ABB RAPID module: Operations.mod

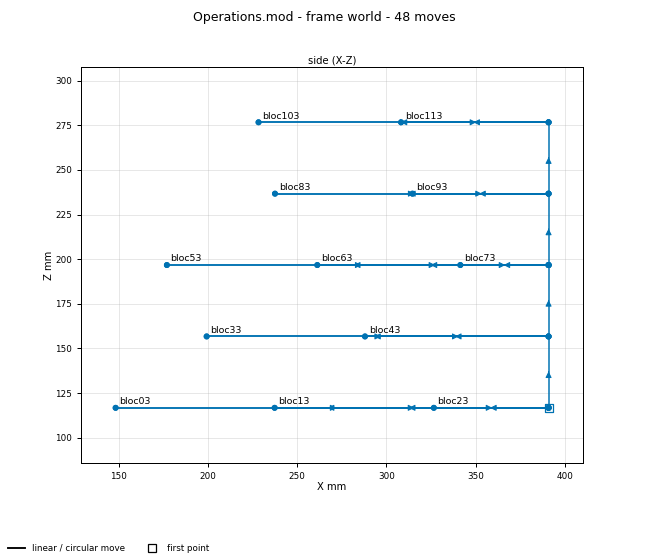
[picture p0: tool path of Operations.mod in frame world, 48 of 49 moves have a stored position in this frame; points joined in program order, loops and branches not executed]
MODULE Operations
 PROC GoHome()
  !
  VAR speeddata HomeSpeed:=[800,100,5000,1000];
  CONST jointtarget HomeTargets0:=[[19.79,37.43,-27.03,0,79.6,44.79],[0,9E9,9E9,9E9,9E9,9E9]];
  MoveAbsJ HomeTargets0,HomeSpeed,z1,EGP_40_N_N_B;
 ENDPROC
 PROC BuildWall()
  !
  VAR zonedata TransportZone:=[FALSE,5,7.5,7.5,0.75,7.5,0.75];
  VAR speeddata PickSpeed:=[60,100,5000,1000];
  CONST robtarget bloc00:=[[16.37,284,122.19],[-0.2706,-0.6533,0.6533,0.2706],[0,0,-1,0],[0,9E9,9E9,9E9,9E9,9E9]];
  CONST robtarget bloc01:=[[-54.35,284,51.47],[-0.2706,-0.6533,0.6533,0.2706],[0,0,-1,0],[0,9E9,9E9,9E9,9E9,9E9]];
  CONST robtarget bloc02:=[[390.93,-147.52,116.72],[0,-0.5676,0.8233,0],[-1,0,-1,0],[0,9E9,9E9,9E9,9E9,9E9]];
  CONST robtarget bloc03:=[[148.33,-147.52,116.72],[0,-0.5676,0.8233,0],[-1,0,-1,0],[0,9E9,9E9,9E9,9E9,9E9]];
  CONST robtarget bloc04:=[[148.33,-263.37,116.72],[0,-0.5676,0.8233,0],[-1,0,-2,0],[0,9E9,9E9,9E9,9E9,9E9]];
  CONST robtarget bloc05:=[[148.33,-263.37,16.72],[0,-0.5676,0.8233,0],[-1,0,-2,0],[0,9E9,9E9,9E9,9E9,9E9]];
  CONST robtarget bloc10:=[[16.37,284,122.19],[-0.2706,-0.6533,0.6533,0.2706],[0,0,-1,0],[0,9E9,9E9,9E9,9E9,9E9]];
  CONST robtarget bloc11:=[[-54.35,284,51.47],[-0.2706,-0.6533,0.6533,0.2706],[0,0,-1,0],[0,9E9,9E9,9E9,9E9,9E9]];
  CONST robtarget bloc12:=[[390.93,-147.52,116.72],[0,-0.6609,0.7505,0],[-1,0,-1,0],[0,9E9,9E9,9E9,9E9,9E9]];
  CONST robtarget bloc13:=[[237.43,-147.52,116.72],[0,-0.6609,0.7505,0],[-1,0,-1,0],[0,9E9,9E9,9E9,9E9,9E9]];
  CONST robtarget bloc14:=[[237.43,-286.18,116.72],[0,-0.6609,0.7505,0],[-1,0,-2,0],[0,9E9,9E9,9E9,9E9,9E9]];
  CONST robtarget bloc15:=[[237.43,-286.18,16.72],[0,-0.6609,0.7505,0],[-1,0,-2,0],[0,9E9,9E9,9E9,9E9,9E9]];
  CONST robtarget bloc20:=[[16.37,284,122.19],[-0.2706,-0.6533,0.6533,0.2706],[0,0,-1,0],[0,9E9,9E9,9E9,9E9,9E9]];
  CONST robtarget bloc21:=[[-54.35,284,51.47],[-0.2706,-0.6533,0.6533,0.2706],[0,0,-1,0],[0,9E9,9E9,9E9,9E9,9E9]];
  CONST robtarget bloc22:=[[390.93,-147.52,116.72],[0,0.7222,-0.6917,0],[-1,0,-1,0],[0,9E9,9E9,9E9,9E9,9E9]];
  CONST robtarget bloc23:=[[326.64,-147.52,116.72],[0,0.7222,-0.6917,0],[-1,0,-2,0],[0,9E9,9E9,9E9,9E9,9E9]];
  CONST robtarget bloc24:=[[326.64,-289.82,116.72],[0,0.7222,-0.6917,0],[-1,0,-2,0],[0,9E9,9E9,9E9,9E9,9E9]];
  CONST robtarget bloc25:=[[326.64,-289.82,16.72],[0,0.7222,-0.6917,0],[-1,0,-2,0],[0,9E9,9E9,9E9,9E9,9E9]];
  CONST robtarget bloc30:=[[16.37,284,122.19],[-0.2706,-0.6533,0.6533,0.2706],[0,0,-1,0],[0,9E9,9E9,9E9,9E9,9E9]];
  CONST robtarget bloc31:=[[-54.35,284,51.47],[-0.2706,-0.6533,0.6533,0.2706],[0,0,-1,0],[0,9E9,9E9,9E9,9E9,9E9]];
  CONST robtarget bloc32:=[[390.93,-147.52,156.72],[0,-0.6058,0.7956,0],[-1,0,-1,0],[0,9E9,9E9,9E9,9E9,9E9]];
  CONST robtarget bloc33:=[[199.33,-147.52,156.72],[0,-0.6058,0.7956,0],[-1,0,-1,0],[0,9E9,9E9,9E9,9E9,9E9]];
  CONST robtarget bloc34:=[[199.33,-268.81,156.72],[0,-0.6058,0.7956,0],[-1,0,-2,0],[0,9E9,9E9,9E9,9E9,9E9]];
  CONST robtarget bloc35:=[[199.33,-268.81,56.72],[0,-0.6058,0.7956,0],[-1,0,-2,0],[0,9E9,9E9,9E9,9E9,9E9]];
  CONST robtarget bloc40:=[[16.37,284,122.19],[-0.2706,-0.6533,0.6533,0.2706],[0,0,-1,0],[0,9E9,9E9,9E9,9E9,9E9]];
  CONST robtarget bloc41:=[[-54.35,284,51.47],[-0.2706,-0.6533,0.6533,0.2706],[0,0,-1,0],[0,9E9,9E9,9E9,9E9,9E9]];
  CONST robtarget bloc42:=[[390.93,-147.52,156.72],[0,-0.6793,0.7339,0],[-1,0,-1,0],[0,9E9,9E9,9E9,9E9,9E9]];
  CONST robtarget bloc43:=[[288.06,-147.52,156.72],[0,-0.6793,0.7339,0],[-1,0,-1,0],[0,9E9,9E9,9E9,9E9,9E9]];
  CONST robtarget bloc44:=[[288.06,-284.33,156.72],[0,-0.6793,0.7339,0],[-1,0,-2,0],[0,9E9,9E9,9E9,9E9,9E9]];
  CONST robtarget bloc45:=[[288.06,-284.33,56.72],[0,-0.6793,0.7339,0],[-1,0,-2,0],[0,9E9,9E9,9E9,9E9,9E9]];
  CONST robtarget bloc50:=[[16.37,284,122.19],[-0.2706,-0.6533,0.6533,0.2706],[0,0,-1,0],[0,9E9,9E9,9E9,9E9,9E9]];
  CONST robtarget bloc51:=[[-54.35,284,51.47],[-0.2706,-0.6533,0.6533,0.2706],[0,0,-1,0],[0,9E9,9E9,9E9,9E9,9E9]];
  CONST robtarget bloc52:=[[390.93,-147.52,196.72],[0,-0.5921,0.8058,0],[-1,0,-1,0],[0,9E9,9E9,9E9,9E9,9E9]];
  CONST robtarget bloc53:=[[177.04,-147.52,196.72],[0,-0.5921,0.8058,0],[-1,0,-1,0],[0,9E9,9E9,9E9,9E9,9E9]];
  CONST robtarget bloc54:=[[177.04,-252.96,196.72],[0,-0.5921,0.8058,0],[-1,0,-2,0],[0,9E9,9E9,9E9,9E9,9E9]];
  CONST robtarget bloc55:=[[177.04,-252.96,96.72],[0,-0.5921,0.8058,0],[-1,0,-2,0],[0,9E9,9E9,9E9,9E9,9E9]];
  CONST robtarget bloc60:=[[16.37,284,122.19],[-0.2706,-0.6533,0.6533,0.2706],[0,0,-1,0],[0,9E9,9E9,9E9,9E9,9E9]];
  CONST robtarget bloc61:=[[-54.35,284,51.47],[-0.2706,-0.6533,0.6533,0.2706],[0,0,-1,0],[0,9E9,9E9,9E9,9E9,9E9]];
  CONST robtarget bloc62:=[[390.93,-147.52,196.72],[0,-0.6476,0.762,0],[-1,0,-1,0],[0,9E9,9E9,9E9,9E9,9E9]];
  CONST robtarget bloc63:=[[261.33,-147.52,196.72],[0,-0.6476,0.762,0],[-1,0,-1,0],[0,9E9,9E9,9E9,9E9,9E9]];
  CONST robtarget bloc64:=[[261.33,-272.79,196.72],[0,-0.6476,0.762,0],[-1,0,-2,0],[0,9E9,9E9,9E9,9E9,9E9]];
  CONST robtarget bloc65:=[[261.33,-272.79,96.72],[0,-0.6476,0.762,0],[-1,0,-2,0],[0,9E9,9E9,9E9,9E9,9E9]];
  CONST robtarget bloc70:=[[16.37,284,122.19],[-0.2706,-0.6533,0.6533,0.2706],[0,0,-1,0],[0,9E9,9E9,9E9,9E9,9E9]];
  CONST robtarget bloc71:=[[-54.35,284,51.47],[-0.2706,-0.6533,0.6533,0.2706],[0,0,-1,0],[0,9E9,9E9,9E9,9E9,9E9]];
  CONST robtarget bloc72:=[[390.93,-147.52,196.72],[0,0.7159,-0.6982,0],[-1,0,-1,0],[0,9E9,9E9,9E9,9E9,9E9]];
  CONST robtarget bloc73:=[[341.48,-147.52,196.72],[0,0.7159,-0.6982,0],[-1,0,-1,0],[0,9E9,9E9,9E9,9E9,9E9]];
  CONST robtarget bloc74:=[[341.48,-279.04,196.72],[0,0.7159,-0.6982,0],[-1,0,-2,0],[0,9E9,9E9,9E9,9E9,9E9]];
  CONST robtarget bloc75:=[[341.48,-279.04,96.72],[0,0.7159,-0.6982,0],[-1,0,-2,0],[0,9E9,9E9,9E9,9E9,9E9]];
  CONST robtarget bloc80:=[[16.37,284,122.19],[-0.2706,-0.6533,0.6533,0.2706],[0,0,-1,0],[0,9E9,9E9,9E9,9E9,9E9]];
  CONST robtarget bloc81:=[[-54.35,284,51.47],[-0.2706,-0.6533,0.6533,0.2706],[0,0,-1,0],[0,9E9,9E9,9E9,9E9,9E9]];
  CONST robtarget bloc82:=[[390.93,-147.52,236.72],[0,-0.6442,0.7648,0],[-1,0,-1,0],[0,9E9,9E9,9E9,9E9,9E9]];
  CONST robtarget bloc83:=[[237.62,-147.52,236.72],[0,-0.6442,0.7648,0],[-1,0,-1,0],[0,9E9,9E9,9E9,9E9,9E9]];
  CONST robtarget bloc84:=[[237.62,-258.84,236.72],[0,-0.6442,0.7648,0],[-1,0,-2,0],[0,9E9,9E9,9E9,9E9,9E9]];
  CONST robtarget bloc85:=[[237.62,-258.84,136.72],[0,-0.6442,0.7648,0],[-1,0,-2,0],[0,9E9,9E9,9E9,9E9,9E9]];
  CONST robtarget bloc90:=[[16.37,284,122.19],[-0.2706,-0.6533,0.6533,0.2706],[0,0,-1,0],[0,9E9,9E9,9E9,9E9,9E9]];
  CONST robtarget bloc91:=[[-54.35,284,51.47],[-0.2706,-0.6533,0.6533,0.2706],[0,0,-1,0],[0,9E9,9E9,9E9,9E9,9E9]];
  CONST robtarget bloc92:=[[390.93,-147.52,236.72],[0,-0.6797,0.7335,0],[-1,0,-1,0],[0,9E9,9E9,9E9,9E9,9E9]];
  CONST robtarget bloc93:=[[314.68,-147.52,236.72],[0,-0.6797,0.7335,0],[-1,0,-1,0],[0,9E9,9E9,9E9,9E9,9E9]];
  CONST robtarget bloc94:=[[314.68,-268.74,236.72],[0,-0.6797,0.7335,0],[-1,0,-2,0],[0,9E9,9E9,9E9,9E9,9E9]];
  CONST robtarget bloc95:=[[314.68,-268.74,136.72],[0,-0.6797,0.7335,0],[-1,0,-2,0],[0,9E9,9E9,9E9,9E9,9E9]];
  CONST robtarget bloc100:=[[16.37,284,122.19],[-0.2706,-0.6533,0.6533,0.2706],[0,0,-1,0],[0,9E9,9E9,9E9,9E9,9E9]];
  CONST robtarget bloc101:=[[-54.35,284,51.47],[-0.2706,-0.6533,0.6533,0.2706],[0,0,-1,0],[0,9E9,9E9,9E9,9E9,9E9]];
  CONST robtarget bloc102:=[[390.93,-147.52,276.72],[0,-0.6905,0.7234,0],[-1,0,-1,0],[0,9E9,9E9,9E9,9E9,9E9]];
  CONST robtarget bloc103:=[[228.41,-147.52,276.72],[0,-0.6905,0.7234,0],[-1,0,-2,0],[0,9E9,9E9,9E9,9E9,9E9]];
  CONST robtarget bloc104:=[[228.41,-249.38,276.72],[0,-0.6905,0.7234,0],[-1,0,-2,0],[0,9E9,9E9,9E9,9E9,9E9]];
  CONST robtarget bloc105:=[[228.41,-249.38,176.72],[0,-0.6905,0.7234,0],[-1,0,-2,0],[0,9E9,9E9,9E9,9E9,9E9]];
  CONST robtarget bloc110:=[[16.37,284,122.19],[-0.2706,-0.6533,0.6533,0.2706],[0,0,-1,0],[0,9E9,9E9,9E9,9E9,9E9]];
  CONST robtarget bloc111:=[[-54.35,284,51.47],[-0.2706,-0.6533,0.6533,0.2706],[0,0,-1,0],[0,9E9,9E9,9E9,9E9,9E9]];
  CONST robtarget bloc112:=[[390.93,-147.52,276.72],[0,-0.6849,0.7286,0],[-1,0,-1,0],[0,9E9,9E9,9E9,9E9,9E9]];
  CONST robtarget bloc113:=[[308.27,-147.52,276.72],[0,-0.6849,0.7286,0],[-1,0,-1,0],[0,9E9,9E9,9E9,9E9,9E9]];
  CONST robtarget bloc114:=[[308.27,-253.64,276.72],[0,-0.6849,0.7286,0],[-1,0,-2,0],[0,9E9,9E9,9E9,9E9,9E9]];
  CONST robtarget bloc115:=[[308.27,-253.64,176.72],[0,-0.6849,0.7286,0],[-1,0,-2,0],[0,9E9,9E9,9E9,9E9,9E9]];
  CONST robtarget NNCTarget0:=[[0,0,101],[0,0,1,0],[0,0,1,0],[0,9E9,9E9,9E9,9E9,9E9]];
  CONST robtarget NNCTarget1:=[[0,0,100],[0,0,1,0],[0,0,1,0],[0,9E9,9E9,9E9,9E9,9E9]];
  CONST robtarget NNCTarget2:=[[0,0,15],[0,0,1,0],[0,0,1,0],[0,9E9,9E9,9E9,9E9,9E9]];
  CONST robtarget CalibTarget0:=[[-8.38,284,196.43],[-0.2706,-0.6533,0.6533,0.2706],[0,0,-1,0],[0,9E9,9E9,9E9,9E9,9E9]];
  CONST robtarget CalibTarget1:=[[-100.31,284,104.51],[-0.2706,-0.6533,0.6533,0.2706],[0,0,-1,0],[0,9E9,9E9,9E9,9E9,9E9]];
  VAR speeddata TransportSpeed:=[800,100,5000,1000];
  StartGripper;
  PathAccLim TRUE \AccMax:=0.7, TRUE \DecelMax:=0.7;
  FindBlock EGP_40_N_N_B, NNCTarget0, TransportSpeed;
  TakeBloc NNCTarget1, NNCTarget2, EGP_40_N_N_B, TransportSpeed, PickSpeed, blockWobj;
  GoHome;
  ReleaseBloc CalibTarget0, CalibTarget1, EGP_40_N_N_B, TransportSpeed, PickSpeed, WObj0;
  TakeBloc bloc00, bloc01, EGP_40_N_N_B, TransportSpeed, PickSpeed, WObj0;
  GoHome;
  MoveL bloc02,TransportSpeed,TransportZone,EGP_40_N_N_B\WObj:=WObj0;
  MoveL bloc03,TransportSpeed,TransportZone,EGP_40_N_N_B\WObj:=WObj0;
  ReleaseBloc bloc04, bloc05, EGP_40_N_N_B, TransportSpeed, PickSpeed, WObj0;
  MoveL bloc03,TransportSpeed,TransportZone,EGP_40_N_N_B\WObj:=WObj0;
  MoveL bloc02,TransportSpeed,TransportZone,EGP_40_N_N_B\WObj:=WObj0;
  FindBlock EGP_40_N_N_B, NNCTarget0, TransportSpeed;
  TakeBloc NNCTarget1, NNCTarget2, EGP_40_N_N_B, TransportSpeed, PickSpeed, blockWobj;
  GoHome;
  ReleaseBloc CalibTarget0, CalibTarget1, EGP_40_N_N_B, TransportSpeed, PickSpeed, WObj0;
  TakeBloc bloc10, bloc11, EGP_40_N_N_B, TransportSpeed, PickSpeed, WObj0;
  GoHome;
  MoveL bloc12,TransportSpeed,TransportZone,EGP_40_N_N_B\WObj:=WObj0;
  MoveL bloc13,TransportSpeed,TransportZone,EGP_40_N_N_B\WObj:=WObj0;
  ReleaseBloc bloc14, bloc15, EGP_40_N_N_B, TransportSpeed, PickSpeed, WObj0;
  MoveL bloc13,TransportSpeed,TransportZone,EGP_40_N_N_B\WObj:=WObj0;
  MoveL bloc12,TransportSpeed,TransportZone,EGP_40_N_N_B\WObj:=WObj0;
  FindBlock EGP_40_N_N_B, NNCTarget0, TransportSpeed;
  TakeBloc NNCTarget1, NNCTarget2, EGP_40_N_N_B, TransportSpeed, PickSpeed, blockWobj;
  GoHome;
  ReleaseBloc CalibTarget0, CalibTarget1, EGP_40_N_N_B, TransportSpeed, PickSpeed, WObj0;
  TakeBloc bloc20, bloc21, EGP_40_N_N_B, TransportSpeed, PickSpeed, WObj0;
  GoHome;
  MoveL bloc22,TransportSpeed,TransportZone,EGP_40_N_N_B\WObj:=WObj0;
  MoveL bloc23,TransportSpeed,TransportZone,EGP_40_N_N_B\WObj:=WObj0;
  ReleaseBloc bloc24, bloc25, EGP_40_N_N_B, TransportSpeed, PickSpeed, WObj0;
  MoveL bloc23,TransportSpeed,TransportZone,EGP_40_N_N_B\WObj:=WObj0;
  MoveL bloc22,TransportSpeed,TransportZone,EGP_40_N_N_B\WObj:=WObj0;
  FindBlock EGP_40_N_N_B, NNCTarget0, TransportSpeed;
  TakeBloc NNCTarget1, NNCTarget2, EGP_40_N_N_B, TransportSpeed, PickSpeed, blockWobj;
  GoHome;
  ReleaseBloc CalibTarget0, CalibTarget1, EGP_40_N_N_B, TransportSpeed, PickSpeed, WObj0;
  TakeBloc bloc30, bloc31, EGP_40_N_N_B, TransportSpeed, PickSpeed, WObj0;
  GoHome;
  MoveL bloc32,TransportSpeed,TransportZone,EGP_40_N_N_B\WObj:=WObj0;
  MoveL bloc33,TransportSpeed,TransportZone,EGP_40_N_N_B\WObj:=WObj0;
  ReleaseBloc bloc34, bloc35, EGP_40_N_N_B, TransportSpeed, PickSpeed, WObj0;
  MoveL bloc33,TransportSpeed,TransportZone,EGP_40_N_N_B\WObj:=WObj0;
  MoveL bloc32,TransportSpeed,TransportZone,EGP_40_N_N_B\WObj:=WObj0;
  FindBlock EGP_40_N_N_B, NNCTarget0, TransportSpeed;
  TakeBloc NNCTarget1, NNCTarget2, EGP_40_N_N_B, TransportSpeed, PickSpeed, blockWobj;
  GoHome;
  ReleaseBloc CalibTarget0, CalibTarget1, EGP_40_N_N_B, TransportSpeed, PickSpeed, WObj0;
  TakeBloc bloc40, bloc41, EGP_40_N_N_B, TransportSpeed, PickSpeed, WObj0;
  GoHome;
  MoveL bloc42,TransportSpeed,TransportZone,EGP_40_N_N_B\WObj:=WObj0;
  MoveL bloc43,TransportSpeed,TransportZone,EGP_40_N_N_B\WObj:=WObj0;
  ReleaseBloc bloc44, bloc45, EGP_40_N_N_B, TransportSpeed, PickSpeed, WObj0;
  MoveL bloc43,TransportSpeed,TransportZone,EGP_40_N_N_B\WObj:=WObj0;
  MoveL bloc42,TransportSpeed,TransportZone,EGP_40_N_N_B\WObj:=WObj0;
  FindBlock EGP_40_N_N_B, NNCTarget0, TransportSpeed;
  TakeBloc NNCTarget1, NNCTarget2, EGP_40_N_N_B, TransportSpeed, PickSpeed, blockWobj;
  GoHome;
  ReleaseBloc CalibTarget0, CalibTarget1, EGP_40_N_N_B, TransportSpeed, PickSpeed, WObj0;
  TakeBloc bloc50, bloc51, EGP_40_N_N_B, TransportSpeed, PickSpeed, WObj0;
  GoHome;
  MoveL bloc52,TransportSpeed,TransportZone,EGP_40_N_N_B\WObj:=WObj0;
  MoveL bloc53,TransportSpeed,TransportZone,EGP_40_N_N_B\WObj:=WObj0;
  ReleaseBloc bloc54, bloc55, EGP_40_N_N_B, TransportSpeed, PickSpeed, WObj0;
  MoveL bloc53,TransportSpeed,TransportZone,EGP_40_N_N_B\WObj:=WObj0;
  MoveL bloc52,TransportSpeed,TransportZone,EGP_40_N_N_B\WObj:=WObj0;
  FindBlock EGP_40_N_N_B, NNCTarget0, TransportSpeed;
  TakeBloc NNCTarget1, NNCTarget2, EGP_40_N_N_B, TransportSpeed, PickSpeed, blockWobj;
  GoHome;
  ReleaseBloc CalibTarget0, CalibTarget1, EGP_40_N_N_B, TransportSpeed, PickSpeed, WObj0;
  TakeBloc bloc60, bloc61, EGP_40_N_N_B, TransportSpeed, PickSpeed, WObj0;
  GoHome;
  MoveL bloc62,TransportSpeed,TransportZone,EGP_40_N_N_B\WObj:=WObj0;
  MoveL bloc63,TransportSpeed,TransportZone,EGP_40_N_N_B\WObj:=WObj0;
  ReleaseBloc bloc64, bloc65, EGP_40_N_N_B, TransportSpeed, PickSpeed, WObj0;
  MoveL bloc63,TransportSpeed,TransportZone,EGP_40_N_N_B\WObj:=WObj0;
  MoveL bloc62,TransportSpeed,TransportZone,EGP_40_N_N_B\WObj:=WObj0;
  FindBlock EGP_40_N_N_B, NNCTarget0, TransportSpeed;
  TakeBloc NNCTarget1, NNCTarget2, EGP_40_N_N_B, TransportSpeed, PickSpeed, blockWobj;
  GoHome;
  ReleaseBloc CalibTarget0, CalibTarget1, EGP_40_N_N_B, TransportSpeed, PickSpeed, WObj0;
  TakeBloc bloc70, bloc71, EGP_40_N_N_B, TransportSpeed, PickSpeed, WObj0;
  GoHome;
  MoveL bloc72,TransportSpeed,TransportZone,EGP_40_N_N_B\WObj:=WObj0;
  MoveL bloc73,TransportSpeed,TransportZone,EGP_40_N_N_B\WObj:=WObj0;
  ReleaseBloc bloc74, bloc75, EGP_40_N_N_B, TransportSpeed, PickSpeed, WObj0;
  MoveL bloc73,TransportSpeed,TransportZone,EGP_40_N_N_B\WObj:=WObj0;
  MoveL bloc72,TransportSpeed,TransportZone,EGP_40_N_N_B\WObj:=WObj0;
  FindBlock EGP_40_N_N_B, NNCTarget0, TransportSpeed;
  TakeBloc NNCTarget1, NNCTarget2, EGP_40_N_N_B, TransportSpeed, PickSpeed, blockWobj;
  GoHome;
  ReleaseBloc CalibTarget0, CalibTarget1, EGP_40_N_N_B, TransportSpeed, PickSpeed, WObj0;
  TakeBloc bloc80, bloc81, EGP_40_N_N_B, TransportSpeed, PickSpeed, WObj0;
  GoHome;
  MoveL bloc82,TransportSpeed,TransportZone,EGP_40_N_N_B\WObj:=WObj0;
  MoveL bloc83,TransportSpeed,TransportZone,EGP_40_N_N_B\WObj:=WObj0;
  ReleaseBloc bloc84, bloc85, EGP_40_N_N_B, TransportSpeed, PickSpeed, WObj0;
  MoveL bloc83,TransportSpeed,TransportZone,EGP_40_N_N_B\WObj:=WObj0;
  MoveL bloc82,TransportSpeed,TransportZone,EGP_40_N_N_B\WObj:=WObj0;
  FindBlock EGP_40_N_N_B, NNCTarget0, TransportSpeed;
  TakeBloc NNCTarget1, NNCTarget2, EGP_40_N_N_B, TransportSpeed, PickSpeed, blockWobj;
  GoHome;
  ReleaseBloc CalibTarget0, CalibTarget1, EGP_40_N_N_B, TransportSpeed, PickSpeed, WObj0;
  TakeBloc bloc90, bloc91, EGP_40_N_N_B, TransportSpeed, PickSpeed, WObj0;
  GoHome;
  MoveL bloc92,TransportSpeed,TransportZone,EGP_40_N_N_B\WObj:=WObj0;
  MoveL bloc93,TransportSpeed,TransportZone,EGP_40_N_N_B\WObj:=WObj0;
  ReleaseBloc bloc94, bloc95, EGP_40_N_N_B, TransportSpeed, PickSpeed, WObj0;
  MoveL bloc93,TransportSpeed,TransportZone,EGP_40_N_N_B\WObj:=WObj0;
  MoveL bloc92,TransportSpeed,TransportZone,EGP_40_N_N_B\WObj:=WObj0;
  FindBlock EGP_40_N_N_B, NNCTarget0, TransportSpeed;
  TakeBloc NNCTarget1, NNCTarget2, EGP_40_N_N_B, TransportSpeed, PickSpeed, blockWobj;
  GoHome;
  ReleaseBloc CalibTarget0, CalibTarget1, EGP_40_N_N_B, TransportSpeed, PickSpeed, WObj0;
  TakeBloc bloc100, bloc101, EGP_40_N_N_B, TransportSpeed, PickSpeed, WObj0;
  GoHome;
  MoveL bloc102,TransportSpeed,TransportZone,EGP_40_N_N_B\WObj:=WObj0;
  MoveL bloc103,TransportSpeed,TransportZone,EGP_40_N_N_B\WObj:=WObj0;
  ReleaseBloc bloc104, bloc105, EGP_40_N_N_B, TransportSpeed, PickSpeed, WObj0;
  MoveL bloc103,TransportSpeed,TransportZone,EGP_40_N_N_B\WObj:=WObj0;
  MoveL bloc102,TransportSpeed,TransportZone,EGP_40_N_N_B\WObj:=WObj0;
  FindBlock EGP_40_N_N_B, NNCTarget0, TransportSpeed;
  TakeBloc NNCTarget1, NNCTarget2, EGP_40_N_N_B, TransportSpeed, PickSpeed, blockWobj;
  GoHome;
  ReleaseBloc CalibTarget0, CalibTarget1, EGP_40_N_N_B, TransportSpeed, PickSpeed, WObj0;
  TakeBloc bloc110, bloc111, EGP_40_N_N_B, TransportSpeed, PickSpeed, WObj0;
  GoHome;
  MoveL bloc112,TransportSpeed,TransportZone,EGP_40_N_N_B\WObj:=WObj0;
  MoveL bloc113,TransportSpeed,TransportZone,EGP_40_N_N_B\WObj:=WObj0;
  ReleaseBloc bloc114, bloc115, EGP_40_N_N_B, TransportSpeed, PickSpeed, WObj0;
  MoveL bloc113,TransportSpeed,TransportZone,EGP_40_N_N_B\WObj:=WObj0;
  MoveL bloc112,TransportSpeed,TransportZone,EGP_40_N_N_B\WObj:=WObj0;
  ShutdownGripper;
 ENDPROC
ENDMODULE
